Fanuc TP program (LS listing): usspulsecnt.ls

/PROG  USSPULSECNT
/ATTR
OWNER		= MNEDITOR;
COMMENT		= "";
PROG_SIZE	= 148;
CREATE		= DATE 20-04-07  TIME 22:58:46;
MODIFIED	= DATE 20-04-08  TIME 04:40:44;
FILE_NAME	= ;
VERSION		= 0;
LINE_COUNT	= 1;
MEMORY_SIZE	= 516;
PROTECT		= READ_WRITE;
TCD:  STACK_SIZE	= 0,
      TASK_PRIORITY	= 50,
      TIME_SLICE	= 0,
      BUSY_LAMP_OFF	= 0,
      ABORT_REQUEST	= 0,
      PAUSE_REQUEST	= 7;
DEFAULT_GROUP	= *,*,*,*,*;
CONTROL_CODE	= 00000000 00000000;
/MN
   1:  R[13]=1    ;
/POS
/END
